// Mitsubishi GX Works2 project: 分拣站   PLC: FX3U/FX3UC

PROGRAM MAIN
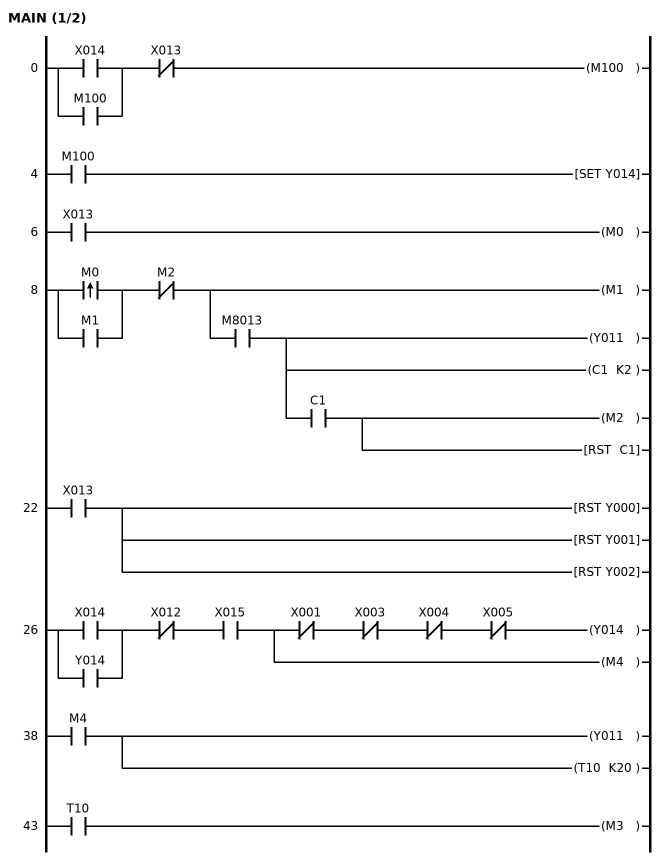
0     LD      X014
      OR      M100
      ANI     X013
      OUT     M100
4     LD      M100
      SET     Y014
6     LD      X013
      OUT     M0
8     LDP     M0
      OR      M1
      ANI     M2
      OUT     M1
      AND     M8013
      OUT     Y011
      OUT     C1 K2
      AND     C1
      OUT     M2
      RST     C1
22    LD      X013
      RST     Y000
      RST     Y001
      RST     Y002
26    LD      X014
      OR      Y014
      ANI     X012
      AND     X015
      MPS
      ANI     X001
      ANI     X003
      ANI     X004
      ANI     X005
      OUT     Y014
      MPP
      OUT     M4
38    LD      M4
      OUT     Y011
      OUT     T10 K20
43    LD      T10
      OUT     M3
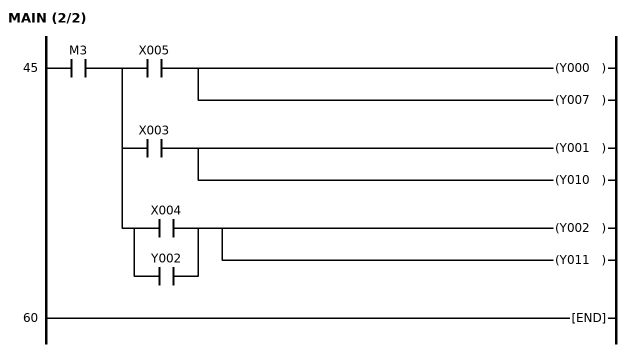
45    LD      M3
      MPS
      AND     X005
      OUT     Y000
      OUT     Y007
      MRD
      AND     X003
      OUT     Y001
      OUT     Y010
      MPP
      LD      X004
      OR      Y002
      ANB
      OUT     Y002
      OUT     Y011
60    END
END_PROGRAM
